SUBAPPLICATION Uebung_126b2 (* Übung zu ISOBUS Send Message Cyclic (mit CB) SINUS-Funktion Plotten *)
  (* Standard: 61499-2; Description: Copyright (c) 2023 Meisterschulen am Ostbahnhof This program and the accompanying materials are made available under the terms of the Eclipse Public License 2.0 which is available at https://www.eclipse.org/legal/epl-2.0/ SPDX-License-Identifier: EPL-2.0 *)
  (* Version 1.0, 2023-10-23, Franz Höpfinger, Meisterschulen am Ostbahnhof, initial API and implementation and/or initial documentation *)
  PACKAGE Uebungen;
  IMPORT Uebungen::const::Uebung_120_129::Filter::PEAK_ADD;
  IMPORT Uebungen::const::Uebung_120_129::Filter::PEAK_FLT;
  IMPORT isobus::pgn::ISOUSERHOME_e::network;
  IMPORT isobus::pgn::ISO_CAN_NODE::NODE1;
  IMPORT isobus::pgn::const::PgnDef::PGN_PDU1_PropA;
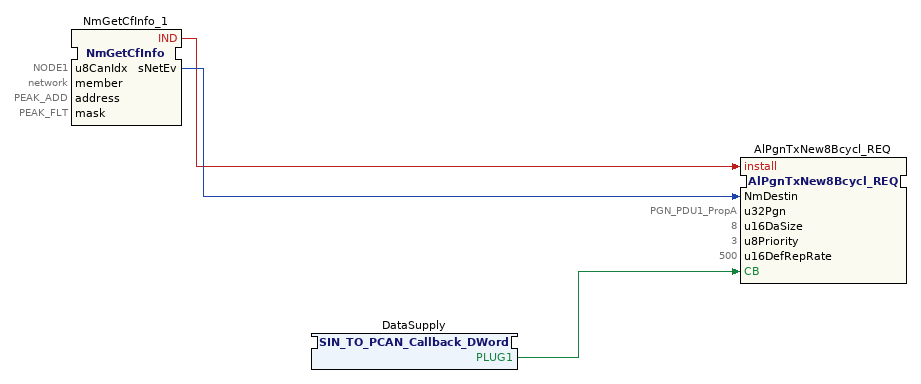
  FBS
    NmGetCfInfo_1 : isobus::pgn::NmGetCfInfo(u8CanIdx := NODE1, member := network, address := PEAK_ADD, mask := PEAK_FLT);
    AlPgnTxNew8Bcycl_REQ : isobus::pgn::tx::AlPgnTxNew8Bcycl_REQ(u32Pgn := PGN_PDU1_PropA, u16DaSize := 8, u8Priority := 3, u16DefRepRate := 500);
  END_FBS
  SUBAPPS
    DataSupply : MyLib::sys::SIN_TO_PCAN_Callback_DWord;
  END_SUBAPPS
  EVENT_CONNECTIONS
    NmGetCfInfo_1.IND TO AlPgnTxNew8Bcycl_REQ.install;
  END_CONNECTIONS
  DATA_CONNECTIONS
    NmGetCfInfo_1.sNetEv TO AlPgnTxNew8Bcycl_REQ.NmDestin;
  END_CONNECTIONS
  ADAPTER_CONNECTIONS
    DataSupply.PLUG1 TO AlPgnTxNew8Bcycl_REQ.CB;
  END_CONNECTIONS
END_SUBAPPLICATION
